SYSTEM VAV_MVL (* Variable Air Valve System Model+View+HMI *)
  (* Standard: 61499-1; Classification: Simulation; ApplicationDomain: HVAC *)
  (* Version 0.2, 2006-05-01, JHC, Holobloc Inc, Changed VAV_MVLL.FV to FD. *)
  (* Version 0.1, 2006-04-27, JHC, Holobloc Inc, Added DUCTS.DAMPER_UI. *)
  (* Version 0.0, 2006-04-12, JHC, Holobloc Inc *)
  DEVICE RECORDER : FRAME_DEVICE(BOUNDS := [240,100,210,250])
    RESOURCE RECORDER : PANEL_RESOURCE
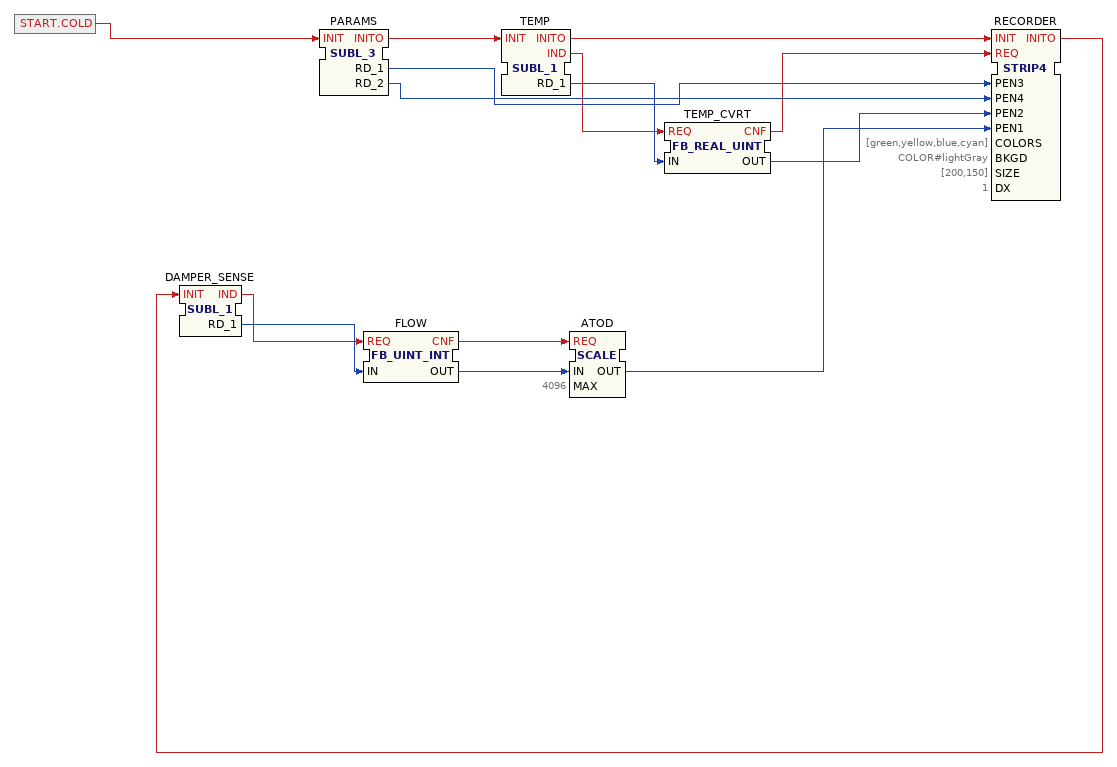
      FBS
        RECORDER : STRIP4(COLORS := [green,yellow,blue,cyan], BKGD := COLOR#lightGray, SIZE := [200,150], DX := 1);
        TEMP : SUBL_1;
        PARAMS : SUBL_3;
        DAMPER_SENSE : SUBL_1;
        TEMP_CVRT : FB_REAL_UINT;
        ATOD : SCALE(MAX := 4096); (* Unscale A/D value *)
        FLOW : FB_UINT_INT;
      END_FBS
      EVENT_CONNECTIONS
        START.COLD TO PARAMS.INIT;
        TEMP.INITO TO RECORDER.INIT;
        TEMP.IND TO TEMP_CVRT.REQ;
        TEMP_CVRT.CNF TO RECORDER.REQ;
        PARAMS.INITO TO TEMP.INIT;
        RECORDER.INITO TO DAMPER_SENSE.INIT;
        DAMPER_SENSE.IND TO FLOW.REQ;
        FLOW.CNF TO ATOD.REQ;
      END_CONNECTIONS
      DATA_CONNECTIONS
        PARAMS.RD_1 TO RECORDER.PEN3;
        PARAMS.RD_2 TO RECORDER.PEN4;
        TEMP.RD_1 TO TEMP_CVRT.IN;
        TEMP_CVRT.OUT TO RECORDER.PEN2;
        ATOD.OUT TO RECORDER.PEN1;
        FLOW.OUT TO ATOD.IN;
        DAMPER_SENSE.RD_1 TO FLOW.IN;
      END_CONNECTIONS
    END_RESOURCE
    RESOURCE PARAMS : PANEL_RESOURCE(ROWS := 2, COLS := 2)
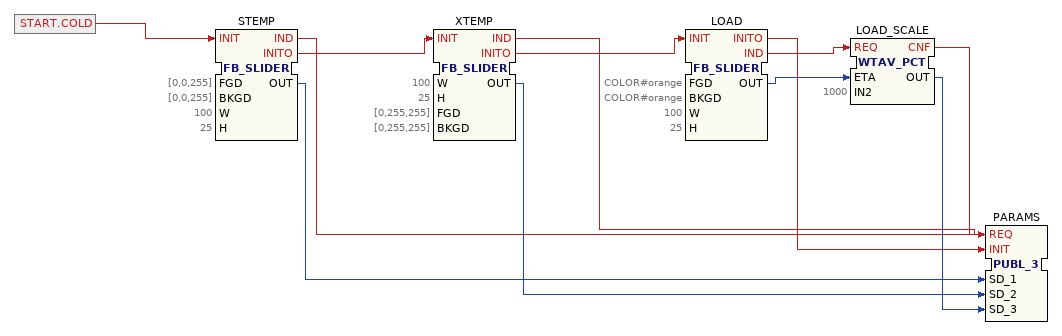
      FBS
        PARAMS : PUBL_3;
        STEMP : FB_SLIDER(FGD := [0,0,255], BKGD := [0,0,255], W := 100, H := 25);
        XTEMP : FB_SLIDER(W := 100, H := 25, FGD := [0,255,255], BKGD := [0,255,255]);
        LOAD : FB_SLIDER(FGD := COLOR#orange, BKGD := COLOR#orange, W := 100, H := 25);
        LOAD_SCALE : WTAV_PCT(IN2 := 1000);
      END_FBS
      EVENT_CONNECTIONS
        STEMP.IND TO PARAMS.REQ;
        STEMP.INITO TO XTEMP.INIT;
        XTEMP.IND TO PARAMS.REQ;
        XTEMP.INITO TO LOAD.INIT;
        LOAD.INITO TO PARAMS.INIT;
        START.COLD TO STEMP.INIT;
        LOAD.IND TO LOAD_SCALE.REQ;
        LOAD_SCALE.CNF TO PARAMS.REQ;
      END_CONNECTIONS
      DATA_CONNECTIONS
        STEMP.OUT TO PARAMS.SD_1;
        XTEMP.OUT TO PARAMS.SD_2;
        LOAD.OUT TO LOAD_SCALE.ETA;
        LOAD_SCALE.OUT TO PARAMS.SD_3;
      END_CONNECTIONS
    END_RESOURCE
  END_DEVICE
  DEVICE CTRL : FRAME_DEVICE(BOUNDS := [100,100,140,270])
    RESOURCE FACE : PANEL_RESOURCE
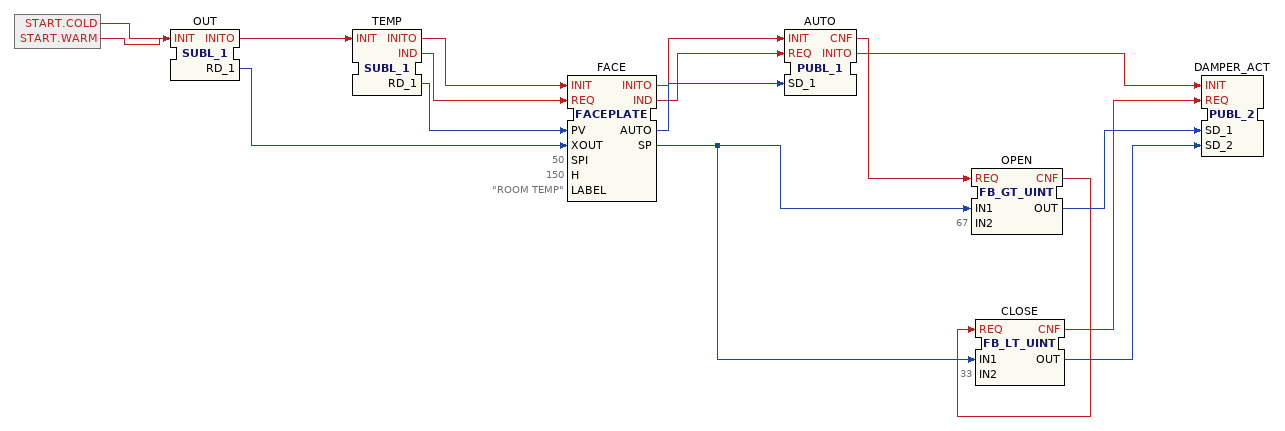
      FBS
        TEMP : SUBL_1;
        FACE : FACEPLATE(SPI := 50, H := 150, LABEL := "ROOM TEMP");
        OUT : SUBL_1;
        AUTO : PUBL_1;
        OPEN : FB_GT_UINT(IN2 := 67);
        CLOSE : FB_LT_UINT(IN2 := 33);
        DAMPER_ACT : PUBL_2;
      END_FBS
      EVENT_CONNECTIONS
        FACE.INITO TO AUTO.INIT;
        FACE.IND TO AUTO.REQ;
        START.COLD TO OUT.INIT;
        START.WARM TO OUT.INIT;
        OUT.INITO TO TEMP.INIT;
        TEMP.INITO TO FACE.INIT;
        TEMP.IND TO FACE.REQ;
        AUTO.CNF TO OPEN.REQ;
        OPEN.CNF TO CLOSE.REQ;
        AUTO.INITO TO DAMPER_ACT.INIT;
        CLOSE.CNF TO DAMPER_ACT.REQ;
      END_CONNECTIONS
      DATA_CONNECTIONS
        TEMP.RD_1 TO FACE.PV;
        OUT.RD_1 TO FACE.XOUT;
        FACE.AUTO TO AUTO.SD_1;
        FACE.SP TO OPEN.IN1;
        FACE.SP TO CLOSE.IN1;
        OPEN.OUT TO DAMPER_ACT.SD_1;
        CLOSE.OUT TO DAMPER_ACT.SD_2;
      END_CONNECTIONS
    END_RESOURCE
  END_DEVICE
  DEVICE ZONE : FRAME_DEVICE(BOUNDS := [450,100,290,250])
    RESOURCE MODEL : EMB_RES
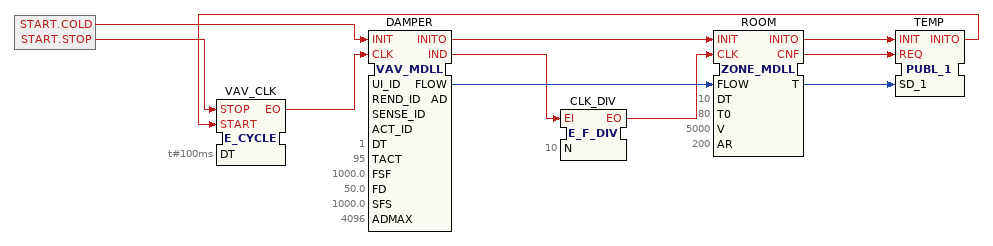
      FBS
        DAMPER : VAV_MDLL(DT := 1, TACT := 95, FSF := 1000.0, FD := 50.0, SFS := 1000.0, ADMAX := 4096);
        ROOM : ZONE_MDLL(DT := 10, T0 := 80, V := 5000, AR := 200);
        CLK_DIV : E_F_DIV(N := 10); (* Zone simulation runs 10x slower than valve sim *)
        VAV_CLK : E_CYCLE(DT := t#100ms);
        TEMP : PUBL_1; (* Main Display clock and Temperature publisher *)
      END_FBS
      EVENT_CONNECTIONS
        START.COLD TO DAMPER.INIT;
        DAMPER.INITO TO ROOM.INIT;
        DAMPER.IND TO CLK_DIV.EI;
        CLK_DIV.EO TO ROOM.CLK;
        START.STOP TO VAV_CLK.STOP;
        VAV_CLK.EO TO DAMPER.CLK;
        ROOM.INITO TO TEMP.INIT;
        TEMP.INITO TO VAV_CLK.START;
        ROOM.CNF TO TEMP.REQ;
      END_CONNECTIONS
      DATA_CONNECTIONS
        DAMPER.FLOW TO ROOM.FLOW;
        ROOM.T TO TEMP.SD_1;
      END_CONNECTIONS
    END_RESOURCE
    RESOURCE DUCTS : VIEW_PANEL(DIA := 25, SIZE := [3,8], VERTICAL := 1)
      FBS
        DAMPER_REND : SUBL_1;
        DAMPER : MECH_VIEW(BKGD := [0,0,255], DIR := 0, STYLE := VSTYLE#DAMPER, WKPC := [0,255,0], LEN := 3);
        LBLS : XSPACE(LBLS := ["","===>","","",""], DIMS := [3,6], COLORS := [green,white]);
        OUTLET : XSPACE(COLORS := [yellow,blue], DIMS := [3,1], LBLS := ["","","","","<==="]);
        DAMPER_UI : PUBL_1;
      END_FBS
      EVENT_CONNECTIONS
        START.COLD TO DAMPER_REND.INIT;
        DAMPER_REND.INITO TO DAMPER.INIT;
        DAMPER_REND.IND TO DAMPER.REQ;
        LBLS.INITO TO OUTLET.INIT;
        DAMPER.INITO TO DAMPER_UI.INIT;
        DAMPER.IND TO DAMPER_UI.REQ;
        DAMPER_UI.INITO TO LBLS.INIT;
      END_CONNECTIONS
      DATA_CONNECTIONS
        DAMPER_REND.RD_1 TO DAMPER.POS;
        DAMPER.FAULT TO DAMPER_UI.SD_1;
      END_CONNECTIONS
    END_RESOURCE
    RESOURCE ROOM : VIEW_PANEL(SIZE := [8,8], DIA := 25)
      FBS
        ROOM : ZONE_VIEWL(FGD := [255,255,0], BKGD := [0,0,255], W := 200, SZ := 14, REND_ID := "DAMPER_REND");
        TEMP : SUBL_1;
      END_FBS
      EVENT_CONNECTIONS
        START.COLD TO TEMP.INIT;
        START.WARM TO TEMP.INIT;
        TEMP.INITO TO ROOM.INIT;
        TEMP.IND TO ROOM.REQ;
      END_CONNECTIONS
      DATA_CONNECTIONS
        TEMP.RD_1 TO ROOM.TEMP;
      END_CONNECTIONS
    END_RESOURCE
  END_DEVICE
END_SYSTEM
